// TIA Portal project "analogPlc" (V15)

(* hardware
DEVICE "S7300/ET200M station_1"  S7-300 station
   slot 0: "Rail_0"  Rail  6ES7 390-1***0-0AA0
   slot 2: "PLC_1"  CPU 314C-2 DP  6ES7 314-6CH04-0AB0  V3.3
      slot 0: "MPI interface_1"  MPI
      slot 1: "DP interface_1"  DP
      slot 2: "DI 24/DO 16_1"  DI24/DO16
      slot 3: "AI 5/AO 2_1"  AI5/AO2
      slot 4: "Count_1"  Counter
      slot 5: "Positioning_1"  Positioning
*)

// ===== PLC "PLC_1"  CPU 314C-2 DP =====

VAR_GLOBAL   // PLC tag table "Default tag table"
   "isUseBiolar" AT %M0.0 : Bool;
   "inSensor" AT %IW752 : Int;
   "HLim" AT %MD10 : Real;
   "LLim" AT %MD14 : Real;
   "Tag_4" AT %MW19 : Word;
   "error" AT %MW18 : Word;
   "Tag_6" AT %MD21 : Real;
   "Tag_7" AT %MW20 : Word;
   "nhietDoCamBien" AT %MD20 : Real;
   "mInSensor" AT %IW2 : Int;
   "start" AT %I0.0 : Bool;
   "Tag_11" AT %M0.1 : Bool;
   "stop" AT %I0.1 : Bool;
   "nhietDoDat" AT %MD24 : Real;
   "OnOffContactor" AT %Q0.0 : Bool;
   "Tag_8" AT %I0.2 : Bool;
   "systemStart" AT %Q0.1 : Bool;
   "on_Contactor" AT %M0.2 : Bool;
   "off_contactor" AT %M0.3 : Bool;
END_VAR

ORGANIZATION_BLOCK "Main"   // OB1, LAD
TITLE = "Main Program Sweep (Cycle)"
{ S7_Optimized_Access := 'FALSE' }
VERSION : 0.1
   VAR_TEMP
      OB1_EV_CLASS : Byte;   // Bits 0-3 = 1 (Coming event), Bits 4-7 = 1 (Event class 1)
      OB1_SCAN_1 : Byte;   // 1 (Cold restart scan 1 of OB 1), 3 (Scan 2-n of OB 1)
      OB1_PRIORITY : Byte;   // Priority of OB Execution
      OB1_OB_NUMBR : Byte;   // 1 (Organization block 1, OB1)
      OB1_RESERVED_1 : Byte;   // Reserved for system
      OB1_RESERVED_2 : Byte;   // Reserved for system
      OB1_PREV_CYCLE : Int;   // Cycle time of previous OB1 scan (milliseconds)
      OB1_MIN_CYCLE : Int;   // Minimum cycle time of OB1 (milliseconds)
      OB1_MAX_CYCLE : Int;   // Maximum cycle time of OB1 (milliseconds)
      OB1_DATE_TIME : Date_And_Time;   // Date and time OB1 started
      useBiolar : Bool;
   END_VAR
BEGIN

REGION Network 1
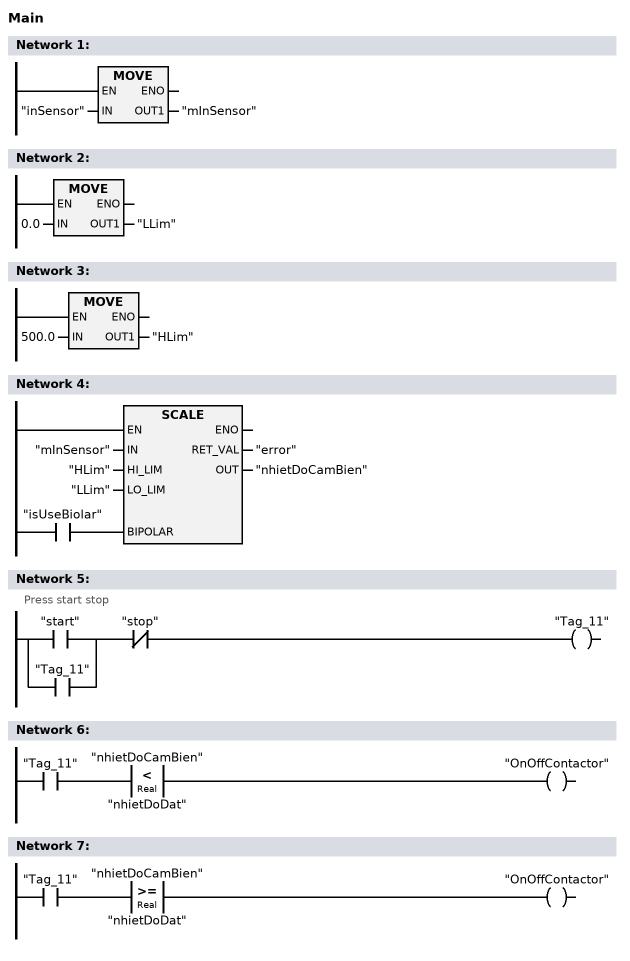
   RUNG wire#powerrail
      { S7_GenerateENO := "TRUE" } Move(in := "inSensor", out1 => "mInSensor")
   END_RUNG
   // the same network as SCL:
   "mInSensor" := "inSensor";
END_REGION

REGION Network 2
   RUNG wire#powerrail
      { S7_GenerateENO := "TRUE" } Move(in := 0.0, out1 => "LLim")
   END_RUNG
   // the same network as SCL:
   "LLim" := 0.0;
END_REGION

REGION Network 3
   RUNG wire#powerrail
      { S7_GenerateENO := "TRUE" } Move(in := 500.0, out1 => "HLim")
   END_RUNG
   // the same network as SCL:
   "HLim" := 500.0;
END_REGION

REGION Network 4
   "error" := SCALE(IN := "mInSensor",
                    HI_LIM := "HLim",
                    LO_LIM := "LLim",
                    BIPOLAR := "isUseBiolar",
                    OUT => "nhietDoCamBien");
END_REGION

REGION Network 5
   // Press start stop
   RUNG wire#powerrail
      Contact( "start" )
      wire#w1
      I_Contact( "stop" )
      Coil( "Tag_11" )
   END_RUNG
   RUNG wire#powerrail
      Contact( "Tag_11" )
   END_RUNG wire#w1
   // the same network as SCL:
   "Tag_11" := ("start" OR "Tag_11") AND NOT "stop";
END_REGION

REGION Network 6
   RUNG wire#powerrail
      Contact( "Tag_11" )
      { S7_Templates := "SrcType := Real" } LT_Contact(in1 := "nhietDoCamBien", in2 := "nhietDoDat")
      Coil( "OnOffContactor" )
   END_RUNG
   // the same network as SCL:
   "OnOffContactor" := "Tag_11" AND ("nhietDoCamBien" < "nhietDoDat");
END_REGION

REGION Network 7
   RUNG wire#powerrail
      Contact( "Tag_11" )
      { S7_Templates := "SrcType := Real" } GE_Contact(in1 := "nhietDoCamBien", in2 := "nhietDoDat")
      Coil( "OnOffContactor" )
   END_RUNG
   // the same network as SCL:
   "OnOffContactor" := "Tag_11" AND ("nhietDoCamBien" >= "nhietDoDat");
END_REGION
END_ORGANIZATION_BLOCK